(* CODESYS project tc3_hbi_utilities.library
   Company: BeckHoff SG
   DefaultNamespace: Tc3_HBI_Utilities
   Version: 3.3.3.1
   Placeholder: Tc3_HBI_Utilities
   Title: Tc3_HBI_Utilities

Project tree, tasks and I/O mapping:
  libraries: Tc2_Standard, * (Beckhoff Automation GmbH); Tc2_System, * (Beckhoff Automation GmbH); Tc2_Utilities, * (Beckhoff Automation GmbH); Tc3_HBI_System, * (Beckhoff)
  BackDoor/
    DUTs/
      data type _ST_BackDoor
      data type _ST_BackDoor_Status
      data type ST_BackDoor
    ITFs/
      interface I_BackDoor
    function block FB_BackDoor_Analog [ST]: M_nBackDoorCtrl
    function block FB_BackDoor_Digital [ST]: M_bBackDoorCtrl
  SafetySensorHandling/
    DUTs/
    ITFs/
      interface I_SensorSignal: M_nControl, M_nOff, P_nAlarmID, P_sAlarmDesc, P_SensorDelay, P_sMessage, P_Timeout
    function block FB_SensorSignal [ST]: M_nControl, M_nOff, M_nReset, P_nAlarmID, P_sAlarmDesc, P_SensorDelay, P_sMessage, P_Timeout
  SignalHandling/
    DUTs/
    ITFs/
      interface I_SignalHandling: M_SetOutput
    function block FB_SignalHandling [ST]: M_SetOutput
    function block FB_SignalHandlingDelay [ST]: M_SetOutput
  Utilities/
    DUTs/
    ITFs/
    function block FB_Utilities [ST]: M_sGetToken
  Version/
    global variables Global_Version
  Tc3_HBI_Utilities.tmc
*)

// BackDoor/DUTs/_ST_BackDoor
TYPE _ST_BackDoor EXTENDS ST_Basic :
STRUCT
END_STRUCT
END_TYPE

// BackDoor/DUTs/_ST_BackDoor_Status
TYPE _ST_BackDoor_Status EXTENDS ST_Basic_Status :
STRUCT
END_STRUCT
END_TYPE

// BackDoor/DUTs/ST_BackDoor
TYPE ST_BackDoor EXTENDS _ST_BackDoor :
STRUCT
	stStatus: _ST_BackDoor_Status;
END_STRUCT
END_TYPE

// Version/Global_Version
{attribute 'TcGenerated'}
// This function has been automatically generated from the project information.
VAR_GLOBAL CONSTANT
	{attribute 'const_non_replaced'}
	{attribute 'linkalways'}
	stLibVersion_Tc3_HBI_Utilities : ST_LibVersion := (iMajor := 3, iMinor := 3, iBuild := 3, iRevision := 1, sVersion := '3.3.3.1');
END_VAR

// BackDoor/ITFs/I_BackDoor
INTERFACE I_BackDoor EXTENDS I_Basic

END_INTERFACE

// BackDoor/FB_BackDoor_Analog
FUNCTION_BLOCK FB_BackDoor_Analog EXTENDS FB_Basic IMPLEMENTS I_BackDoor
VAR_INPUT
END_VAR
VAR_OUTPUT
END_VAR
VAR
	FB_BackDoorAnalog_M_nBackDoorCtrl_iActual: INT;
	FB_BackDoorAnalog_M_nBackDoorCtrl_iSimu	: INT;
	FB_BackDoorAnalog_M_nBackDoorCtrl_iBackDoor	: INT;
	FB_BackDoorAnalog_M_nBackDoorCtrl_bProductionMode	: BOOL:= TRUE;
	FB_BackDoorAnalog_M_nBackDoorCtrl_bBackDoor		: BOOL:= FALSE;
END_VAR

METHOD PUBLIC M_nBackDoorCtrl : INT
VAR_INPUT
	bProductionMode	: BOOL;
	iActual	: INT;
	iSimu	: INT;
	iBackDoor	: INT;
	bBackDoor	: BOOL;
END_VAR
// Local Variables
	FB_BackDoorAnalog_M_nBackDoorCtrl_bProductionMode:= bProductionMode;
	FB_BackDoorAnalog_M_nBackDoorCtrl_bBackDoor:= bBackDoor;
	
	FB_BackDoorAnalog_M_nBackDoorCtrl_iActual:= iActual;
	FB_BackDoorAnalog_M_nBackDoorCtrl_iSimu:= iSimu;
	FB_BackDoorAnalog_M_nBackDoorCtrl_iBackDoor:= iBackDoor;
	
	
	IF FB_BackDoorAnalog_M_nBackDoorCtrl_bProductionMode THEN
	 M_nBackDoorCtrl:= FB_BackDoorAnalog_M_nBackDoorCtrl_iActual;
		ELSIF FB_BackDoorAnalog_M_nBackDoorCtrl_bBackDoor THEN
			M_nBackDoorCtrl:= FB_BackDoorAnalog_M_nBackDoorCtrl_iBackDoor;
			ELSE M_nBackDoorCtrl:= FB_BackDoorAnalog_M_nBackDoorCtrl_iSimu;
 	END_IF
END_METHOD

END_FUNCTION_BLOCK

// BackDoor/FB_BackDoor_Digital
FUNCTION_BLOCK FB_BackDoor_Digital EXTENDS FB_Basic IMPLEMENTS I_BackDoor
VAR_INPUT
END_VAR
VAR_OUTPUT
END_VAR
VAR
	FB_BackDoorDigital_M_nBackDoorCtrl_bActual: BOOL;
	FB_BackDoorDigital_M_nBackDoorCtrl_bSimu	: BOOL;
	FB_BackDoorDigital_M_nBackDoorCtrl_iBackDoor	: INT;
	FB_BackDoorDigital_M_nBackDoorCtrl_bBackDoor	: BOOL;
	FB_BackDoorDigital_M_nBackDoorCtrl_bProductionMode	: BOOL:= TRUE;
END_VAR

METHOD PUBLIC M_bBackDoorCtrl : BOOL
VAR_INPUT
	bProductionMode: BOOL:= TRUE;;
	bActual	: BOOL;
	bSimu	: BOOL;
	iBackDoor	: INT;
END_VAR
// Local Variables
	FB_BackDoorDigital_M_nBackDoorCtrl_bProductionMode:= bProductionMode;
	
	FB_BackDoorDigital_M_nBackDoorCtrl_bActual:= bActual;
	FB_BackDoorDigital_M_nBackDoorCtrl_bSimu:= bSimu;
	FB_BackDoorDigital_M_nBackDoorCtrl_iBackDoor:= iBackDoor;
	
	CASE FB_BackDoorDigital_M_nBackDoorCtrl_iBackDoor OF 
		0:
			FB_BackDoorDigital_M_nBackDoorCtrl_bBackDoor:= FALSE;
		1:
			FB_BackDoorDigital_M_nBackDoorCtrl_bBackDoor:= TRUE;
		2:
			FB_BackDoorDigital_M_nBackDoorCtrl_bBackDoor:= FALSE;
			
	ELSE FB_BackDoorDigital_M_nBackDoorCtrl_bBackDoor:= FALSE;
		
	END_CASE
	
	IF FB_BackDoorDigital_M_nBackDoorCtrl_bProductionMode THEN
	 	M_bBackDoorCtrl:= FB_BackDoorDigital_M_nBackDoorCtrl_bActual;
		ELSIF FB_BackDoorDigital_M_nBackDoorCtrl_iBackDoor= 1 OR FB_BackDoorDigital_M_nBackDoorCtrl_iBackDoor= 2 THEN
			M_bBackDoorCtrl:= FB_BackDoorDigital_M_nBackDoorCtrl_bBackDoor;
			ELSE M_bBackDoorCtrl:= FB_BackDoorDigital_M_nBackDoorCtrl_bSimu;
 	 END_IF
END_METHOD

END_FUNCTION_BLOCK

// SafetySensorHandling/ITFs/I_SensorSignal
INTERFACE I_SensorSignal EXTENDS I_Basic

METHOD PUBLIC M_nControl : UDINT
VAR_INPUT
	bExecute	: BOOL;
	bSensor	: BOOL;
END_VAR
END_METHOD

METHOD M_nOff : UDINT
VAR_INPUT
END_VAR
END_METHOD

PROPERTY P_nAlarmID : UDINT
SET
END_SET
END_PROPERTY

PROPERTY P_sAlarmDesc : STRING
SET
END_SET
END_PROPERTY

PROPERTY P_SensorDelay : TIME
SET
END_SET
END_PROPERTY

PROPERTY P_sMessage : STRING
GET
END_GET
END_PROPERTY

PROPERTY P_Timeout : TIME
SET
END_SET
END_PROPERTY

END_INTERFACE

// SafetySensorHandling/FB_SensorSignal
FUNCTION_BLOCK FB_SensorSignal EXTENDS FB_Basic IMPLEMENTS I_SensorSignal
VAR_INPUT
END_VAR
VAR_OUTPUT
END_VAR
VAR
	FB_SensorSignal_M_nControl_sMessage	: STRING(80);
	FB_SensorSignal_M_nControl_Timeout	: TIME:= T#5S;
	FB_SensorSignal_M_nControl_SensorDelay	: TIME:= T#0MS;
	FB_SensorSignal_M_nControl_iState: INT;
	FB_SensorSignal_M_nControl_bExecute: BOOL;
	FB_SensorSignal_M_nControl_bSensor: BOOL;
	FB_SensorSignal_M_nControl_fbExecute_R_TRIG: Tc2_Standard.R_TRIG;
	FB_SensorSignal_M_nControl_fbTimeout: Tc2_Standard.TON;
	FB_SensorSignal_M_nControl_fbSensorDelay: Tc2_Standard.TON;
	FB_SensorSignal_M_nControl_nAlarmID: UDINT:= 999;
	FB_SensorSignal_M_nControl_sAlarmDesc: STRING(80):= 'Sensor Error';
END_VAR

//	The result of the method is an unsigned double integer
//	0 = idle 
//	1 = coupled
//	2 = starting
//	3 = running
//	4 = aborted
// 	5 = no hardware connected
// 	6 = Spare
//	7 = pointer or index error
//	8 = mapping error
//	9 = parameter error
//	10 = complete
//	21 = cylinder extend error
// 	22 = cylinder retract error
// 	23 = vacuum on error
// 	24 = vacuum off error
// 	25 = purge on error
// 	26 = purge off error
//  27 = Present sensor error
//  28 = Safety sensor error
//	Any other number = ErrorID
METHOD PUBLIC M_nControl : UDINT
VAR_INPUT
	bExecute	: BOOL;
	bSensor		: BOOL;
END_VAR
// =========================================================
// Local variables
	FB_SensorSignal_M_nControl_bExecute:= bExecute;
	FB_SensorSignal_M_nControl_bSensor:= bSensor;
	
// =========================================================	
	IF _bReset THEN
		IF _bError THEN;
			FB_SensorSignal_M_nControl_sMessage:= '';
			IF FB_SensorSignal_M_nControl_bExecute THEN
				FB_SensorSignal_M_nControl_iState:= 01;
			ELSE 
				FB_SensorSignal_M_nControl_iState:= 00;
			END_IF
		END_IF	
	END_IF	
	
// =========================================================
	FB_SensorSignal_M_nControl_fbExecute_R_TRIG(CLK:= FB_SensorSignal_M_nControl_bExecute, Q=> );
	IF FB_SensorSignal_M_nControl_fbExecute_R_TRIG.Q THEN
		FB_SensorSignal_M_nControl_iState:= 01;
	END_IF
	
// =========================================================	
// State machine

	CASE FB_SensorSignal_M_nControl_iState OF 
		
		00: // Do nothing
			M_nControl:= Tc3_HBI_System.cIDLE;
			
		01: // Reset timer
			M_nControl:= Tc3_HBI_System.cSTARTING;
			
			FB_SensorSignal_M_nControl_fbTimeout(IN:= FALSE, PT:= T#0S);
			FB_SensorSignal_M_nControl_fbSensorDelay(IN:= FALSE, PT:= T#0S,);
			FB_SensorSignal_M_nControl_iState:= 2;
			
		02: // Running
			M_nControl:= Tc3_HBI_System.cRUNNING;
			
			FB_SensorSignal_M_nControl_fbTimeout(IN:= NOT FB_SensorSignal_M_nControl_bSensor, PT:= FB_SensorSignal_M_nControl_Timeout, Q=> , ET=> );
			FB_SensorSignal_M_nControl_fbSensorDelay(IN:= FB_SensorSignal_M_nControl_bSensor, PT:= FB_SensorSignal_M_nControl_SensorDelay, Q=> , ET=> );
			IF _bReset THEN
 				FB_SensorSignal_M_nControl_iState:= FB_SensorSignal_M_nControl_iState-1;
				ELSIF FB_SensorSignal_M_nControl_fbSensorDelay.Q THEN
					FB_SensorSignal_M_nControl_fbSensorDelay(IN:= FALSE, PT:= T#0S,);
					FB_SensorSignal_M_nControl_iState:= 03;
					ELSIF FB_SensorSignal_M_nControl_fbTimeout.Q THEN
						FB_SensorSignal_M_nControl_fbTimeout(IN:= FALSE, PT:= T#0S);
//						M_nError(nErrorID:= FB_SafetySignal_M_nControl_nAlarmID);
//						FB_SafetySignal_M_nControl_sMessage:= CONCAT(CONCAT(UDINT_TO_STRING(FB_SafetySignal_M_nControl_nAlarmID),'>')
//																,CONCAT('>',FB_SafetySignal_M_nControl_sDescription));
						FB_SensorSignal_M_nControl_iState:= 999;
			END_IF
		
		03: // Completed
			M_nControl:= Tc3_HBI_System.cCOMPLETE;
			
			IF NOT FB_SensorSignal_M_nControl_bExecute THEN
				FB_SensorSignal_M_nControl_iState:= 00;
			END_IF
			
		999: // Error state
			M_nControl:= Tc3_HBI_System.cABORTED;
			
			M_nError(nErrorID:= FB_SensorSignal_M_nControl_nAlarmID);
			FB_SensorSignal_M_nControl_sMessage:= CONCAT(CONCAT(UDINT_TO_STRING(FB_SensorSignal_M_nControl_nAlarmID),'>')
													,CONCAT('>',FB_SensorSignal_M_nControl_sAlarmDesc));
			
			FB_SensorSignal_M_nControl_fbTimeout(IN:= FALSE, PT:= T#0S);
			
			IF NOT FB_SensorSignal_M_nControl_bExecute THEN
				FB_SensorSignal_M_nControl_iState:= 00;
			END_IF

	ELSE 
		FB_SensorSignal_M_nControl_iState:= 00;
		
	END_CASE
	
THIS^._bReady:= (M_nControl= Tc3_HBI_System.cCOMPLETE);

// =========================================================
END_METHOD

METHOD M_nOff : UDINT
VAR_INPUT
END_VAR
// =========================================================
	M_nControl(bExecute:= FALSE, bSensor:= FALSE);
	
	M_nOff:= Tc3_HBI_System.cCOMPLETE;
// =========================================================
END_METHOD

//	The result of the method is an unsigned double integer
//	0 = idle 
//	1 = coupled
//	2 = starting
//	3 = running
//	4 = aborted
// 	5 = no hardware connected
//  6 = Spare
//	7 = pointer or index error
//	8 = mapping error
//	9 = parameter error
//	10 = complete
//	Any other number = ErrorID
METHOD PUBLIC M_nReset : UDINT
VAR_INPUT
	bExecute: BOOL;
END_VAR
SUPER^.M_nReset(bExecute);

IF _bReset THEN
	IF _bError THEN
		
		FB_SensorSignal_M_nControl_sMessage:= '';
		
		FB_SensorSignal_M_nControl_fbTimeout(IN:= FALSE, PT:= T#0S);
		FB_SensorSignal_M_nControl_fbSensorDelay(IN:= FALSE, PT:= T#0S,);
		
		FB_SensorSignal_M_nControl_bExecute:= FALSE;
		FB_SensorSignal_M_nControl_fbExecute_R_TRIG(CLK:= FALSE, Q=> );
		FB_SensorSignal_M_nControl_iState:= 0;

	END_IF	
END_IF
END_METHOD

{warning 'add property implementation'}
PROPERTY P_nAlarmID : UDINT
SET
FB_SensorSignal_M_nControl_nAlarmID:= P_nAlarmID;
END_SET
END_PROPERTY

PROPERTY P_sAlarmDesc : STRING
SET
FB_SensorSignal_M_nControl_sAlarmDesc:= P_sAlarmDesc;
END_SET
END_PROPERTY

PROPERTY P_SensorDelay : TIME
SET
FB_SensorSignal_M_nControl_SensorDelay:= P_SensorDelay;
END_SET
END_PROPERTY

{warning 'add property implementation'}
PROPERTY P_sMessage : STRING
GET
P_sMessage:= FB_SensorSignal_M_nControl_sMessage;
END_GET
END_PROPERTY

{warning 'add property implementation'}
PROPERTY P_Timeout : TIME
SET
VAR
	_tPresentDelay: TIME;
END_VAR
FB_SensorSignal_M_nControl_Timeout:= P_Timeout;
END_SET
END_PROPERTY

END_FUNCTION_BLOCK

// SignalHandling/ITFs/I_SignalHandling
INTERFACE I_SignalHandling EXTENDS I_Basic

METHOD M_SetOutput
VAR_INPUT
END_VAR
END_METHOD

END_INTERFACE

// SignalHandling/FB_SignalHandling
FUNCTION_BLOCK FB_SignalHandling IMPLEMENTS I_SignalHandling
VAR_INPUT
	bInput		: BOOL;			// Input signal, e.g. sensor signal, fuse
	bEnable		: BOOL;
END_VAR
VAR_OUTPUT
	bOut		: BOOL;
END_VAR

// =========================================================
;
// =========================================================

METHOD PUBLIC M_SetOutput
VAR_INPUT
END_VAR
// =========================================================
	// Out
	
bOut := bInput AND bEnable;

// =========================================================
END_METHOD

END_FUNCTION_BLOCK

// SignalHandling/FB_SignalHandlingDelay
FUNCTION_BLOCK FB_SignalHandlingDelay EXTENDS FB_SignalHandling
VAR_INPUT
	tDelay			: TIME;
END_VAR
VAR
	bSet			: BOOL;
	fbTimerDelay	: TON;
END_VAR

// =========================================================
;
// =========================================================

METHOD PUBLIC M_SetOutput
VAR_INPUT
END_VAR
// =========================================================
	// Out

IF bEnable AND bInput THEN
	bSet := TRUE;
END_IF

IF bSet THEN
	fbTimerDelay(	IN := TRUE,
					PT := tDelay);
ELSE
	fbTimerDelay(	IN := FALSE);
END_IF

IF fbTimerDelay.Q THEN
	bSet := FALSE;
	
	fbTimerDelay(IN := FALSE);
	
	bOut := TRUE;
ELSE
	bOut := FALSE;
END_IF
			
// =========================================================
END_METHOD

END_FUNCTION_BLOCK

// Utilities/FB_Utilities
FUNCTION_BLOCK FB_Utilities EXTENDS FB_Basic
VAR_INPUT
END_VAR
VAR_OUTPUT
END_VAR
VAR
END_VAR

METHOD PUBLIC M_sGetToken : T_MaxString
VAR_INPUT
	sAllTokens: Tc2_System.T_MaxString;
	nToken: UINT;
  	sDelim: STRING;
END_VAR
VAR
// Temporary Variables 
	pString: POINTER TO STRING;
	nCurTokenLocation: INT;
END_VAR
pString:= ADR(sAllTokens);

IF nToken < 1 OR LEN(sDelim) < 1 THEN
	// Negative OR zeroth token OR empty delimiter strings mean an empty token 
	M_sGetToken:= '';
 	RETURN;
ELSE
	IF nToken = 1 THEN
	// Quickly extract the first token 
	nCurTokenLocation:= FIND(pString^, sDelim);
	   	IF nCurTokenLocation > 1 THEN
	   		M_sGetToken:= LEFT(pString^, nCurTokenLocation - 1);
	   	ELSE
			M_sGetToken:= pString^;
	    END_IF
	ELSE
		// FIND the Nth token 
		REPEAT
			nCurTokenLocation:= FIND(pString^, sDelim);
			IF nCurTokenLocation = 0 THEN
				M_sGetToken:= '';
				RETURN;
			ELSE
				pString:= pString + INT_TO_DWORD(nCurTokenLocation -1) + INT_TO_DWORD(LEN(sDelim));
			END_IF
	
			nToken:= nToken - 1;
			UNTIL nToken = 1
		END_REPEAT;

		// Extract the Nth token (Which is the next token AT this point) 
		nCurTokenLocation:= FIND(pString^, sDelim);
		IF nCurTokenLocation > 0 THEN
			M_sGetToken:= LEFT(pString^, nCurTokenLocation - 1);
			RETURN;
		ELSE
			M_sGetToken:= pString^;
		   	RETURN;
		END_IF
	END_IF
END_IF
END_METHOD

END_FUNCTION_BLOCK
